% RSLogix 500 project PLC1_L2-1b.RSS, saved by version 12.00.00.00 %
PROJECT "UNTITLED"    % processor: Bul.1763 MicroLogix 1100 Series B %

PROGRAM FILES
  LAD 2   2 rungs

DATA FILES
  O0 OUTPUT  5 elements
  I1 INPUT  6 elements
  S2 STATUS  66 elements
  B3 BINARY  1 elements
  T4 TIMER  1 elements
  C5 COUNTER  1 elements
  R6 CONTROL  1 elements
  N7 INTEGER  1 elements
  F8 FLOAT  1 elements

LADDER 2
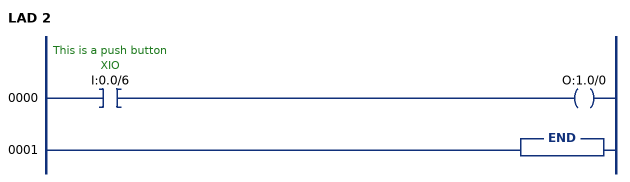
% Rung: 0 %
SOR XIC I:0.0/6 OTE O:1.0/0 EOR
%   I:0.0/6  XIO  "This is a push button" %
% Rung: 1 %
SOR END EOR

OTHER DOCUMENTED ADDRESSES
  I:0.0/0  PB1  "This is Push button 1"
  O:1  LT1  "Light 1"

REVISION NOTES
  0: Completed
  1: test
  2: lab1-1
